(* Basic FB for autodocs tests. *)
FUNCTION_BLOCK FB_Basic
VAR_INPUT
    bEnable : BOOL;
    nValue  : INT := 0;
END_VAR
VAR_OUTPUT
    bDone : BOOL;
END_VAR
VAR_IN_OUT
    stData : ST_TestData;
END_VAR

bDone := bEnable;

END_FUNCTION_BLOCK

(* stored: Version 1.1.0.1
   POU FB_Basic: Id {11111111-1111-1111-1111-111111111101} *)
